TYPE stParamsChamber :
STRUCT
//Nazwy testów / kompresorów
	sTestName 			: STRING := 'Test';			//Nazwa dla aktuanie wykonywanego testu
	sCompressorName 	: STRING;					//Nazwa dla kompresora
	sErrorDescription	: STRING;					//Opis aktualnego błędu
	sChamberName		: STRING;					//Nazwa komory dla zapisu plików
	sFileDirectory		: STRING;					//Lokalizacja dla zapisu plików
	sFileName			: STRING;					//Nazwa pliku
//Konfigruacja komory
	iCompresorType		: nCompresorTypes := 1;			//Typ kompresora
	iTestNumber			: INT;						//Numer testu
	rMinimalPressure	: REAL;						//Ciśnienie minimalne dla startu komory 
	//stChamberTestParams	:s stTestParams;				//Parametry testu dla komory
	//Parametryzacja zapisu plików
	bSaveToFile			: BOOL;						//Czy zezwolić na zapis do pliku
	iSaveEveryRecords	: INT;						//Wykonaj zapis co ile rekodrów
	iSampleTime0_150	: INT;						//Okres próbkowania do zapisu
	iSampleTime0_1		: INT;						//Okres próbkowania do zapisu
	iSampleTime1_x		: INT;						//Okres próbkowania do zapisu
	sFileCopyLocation	: STRING;					//Gdzie kopoiwać pliki

//Struktury do sterowania skalowaniem wartości fizycznych
	stPressureSens 		: stMeasurementScalingData;	// Parametry skalowania prądu
	stVoltageSens 		: stMeasurementScalingData;	// Parametry skalowania napięcia
	stCurrenteSens 		: stMeasurementScalingData;	// Parametry skalowania prądu
END_STRUCT
END_TYPE

(* stored: Version 1.1.0.1, ProductVersion 3.1.4024.12
   DUT stParamsChamber: Id {a772daf8-06a0-49f6-a012-c13d0ba9db5e} *)
